TYPE ST_HomeParams :
STRUCT
  Position              : LREAL;
  HomingMode            : INT;
  Options               : ST_HomingOptionsExt;

  InvertHomeSensor      : BIT := FALSE;   //Set to true,  NormallyClosed home sensor
  SimulateHomeSensor    : BIT := FALSE;   //Set to true,  homed on encoder index only. The homing methode 'hardware sync' must be used then.

  UseLimitMin           : BIT := TRUE;    //Set to false, no negative limit sensor.

  InvertLimitMin        : BIT := FALSE;   //Set to true,  NC negative limit sensor
  HomeOnLimitMin        : BIT := FALSE;   //Set to true,  homed on negative limit sensor 

  UseLimitMax           : BIT := TRUE;    //Set to false, no positive limit sensor.

  InvertLimitMax        : BIT := FALSE;   //Set to true,  NC positive limit sensor
  HomeOnLimitMax        : BIT := FALSE;   //Set to true,  homed on positive limit sensor 
  
  // It is not allowed to use more than 1 of the 3 switches: SimulateHomeSensor, HomeOnLimitMin, HomeOnLimitMax
  
END_STRUCT
END_TYPE

(* stored: Version 1.1.0.1
   DUT ST_HomeParams: Id {fe6817ca-2418-42df-a18e-f69a87736bd6} *)
